// TwinCAT 3 PLC project ads
// ProgramVersion: 3.1.4026.21
// libraries:
//   BufferManager, * (BeckhoffYonatan)
//   Tc2_Standard, * (Beckhoff Automation GmbH)
//   Tc2_System, * (Beckhoff Automation GmbH)
//   Tc2_Utilities, * (Beckhoff Automation GmbH)
// project tree:
//   / PlcTask.TcTTO
//   POUs/ MAIN.TcPOU
// real-time tasks:
//   TASK PlcTask: cycle T#10ms, priority 20, ADS port 350

CONFIGURATION ads
    RESOURCE PLC ON TwinCAT3
        TASK PlcTask(INTERVAL := T#10ms, PRIORITY := 20);
        PROGRAM MAIN WITH PlcTask : MAIN;
    END_RESOURCE
END_CONFIGURATION

// ---- POUs/MAIN.TcPOU
PROGRAM MAIN
VAR
	bBlinker	: BOOL;
	tonBlink	: TON;
	sTime :TIME:= T#1S;
END_VAR


tonBlink(IN := NOT tonBlink.Q, PT := sTime);

IF tonBlink.Q THEN
	bBlinker := NOT bBlinker;
END_IF

END_PROGRAM
